TYPE DigitalOutputBase_1FE0D5EE :
STRUCT
END_STRUCT
END_TYPE

(* stored: Version 1.2.0.0, ProductVersion 3.1.4024.9
   DUT DigitalOutputBase_1FE0D5EE: Id {426b8235-e503-41db-b27e-edddf81a37eb} *)
